// TIA Portal project "Door Locking System" (V17)
// Door Locking System
// When lock button is pressed, the doors should lock and When Unlock button is pressed, the doors remain unlocked for 10s and then unlocked. The doors should not lock if there is someone at the door.

(* hardware
DEVICE "S7-1200 station_1"  S7-1200 Station
   slot 0: "Rack_0"  S7-1200 Rack  Rack  V1.0
   slot 1: "PLC_2"  CPU 1212C AC/DC/Rly  6ES7 212-1BE40-0XB0  V4.5
*)

// ===== PLC "PLC_2"  CPU 1212C AC/DC/Rly =====

VAR_GLOBAL   // PLC tag table "Default tag table"
   "Door Lock Command" AT %I0.0 : Bool;
   "Door Unlock Command" AT %I0.1 : Bool;
   "Door" AT %Q0.0 : Bool;
   "Human_Sensor" AT %I0.2 : Bool;
   "Tag_1" AT %M0.0 : Bool;
   "Tag_2" AT %M0.1 : Bool;
END_VAR

// folder: System blocks/Program resources

DATA_BLOCK "IEC_Timer_0_DB"   // DB1
{ S7_Optimized_Access := 'TRUE' }
AUTHOR : Simatic
FAMILY : IEC
NAME : IEC_TMR
VERSION : 1.0
// stored: InstanceOfName IEC_TIMER
"IEC_TIMER"
BEGIN
END_DATA_BLOCK

// folder: (top level)

ORGANIZATION_BLOCK "Main"   // OB1, LAD, ProgramCycle
TITLE = "Main Program Sweep (Cycle)"
{ S7_Optimized_Access := 'TRUE' }
VERSION : 0.1
   VAR_INPUT
      Initial_Call : Bool;   // Initial call of this OB
      Remanence : Bool;   // =True, if remanent data are available
   END_VAR
BEGIN

REGION Network 2
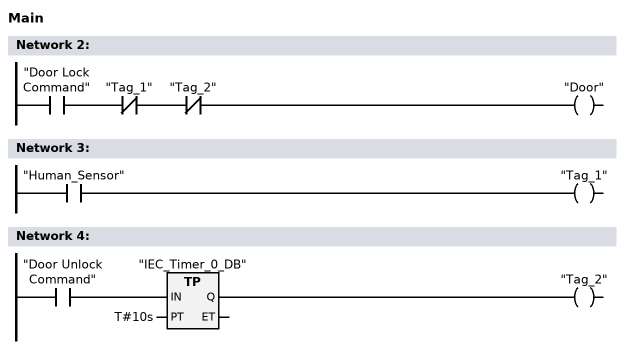
   RUNG wire#powerrail
      Contact( "Door Lock Command" )
      I_Contact( "Tag_1" )
      I_Contact( "Tag_2" )
      Coil( "Door" )
   END_RUNG
   // the same network as SCL:
   "Door" := "Door Lock Command" AND NOT "Tag_1" AND NOT "Tag_2";
END_REGION

REGION Network 3
   RUNG wire#powerrail
      Contact( "Human_Sensor" )
      Coil( "Tag_1" )
   END_RUNG
   // the same network as SCL:
   "Tag_1" := "Human_Sensor";
END_REGION

REGION Network 4
   "IEC_Timer_0_DB".TP(IN := "Door Unlock Command", PT := T#10s);
   "Tag_2" := "IEC_Timer_0_DB".Q;
END_REGION
END_ORGANIZATION_BLOCK